# B&R Automation Studio project Sh_0218_l2
Automation Studio 4.5.2.102

## Configuration labBR

### Task classes (Cpu.sw)
```
Cyclic#4:
  DoorCtrl <- DoorCtrl.prg
  LedCtrl <- LedCtrl.prg
Binaries: TCData, udbdef, ashwd, User, asfw, arconfig, sysconf, Role, iomap, ashwac
Libraries: sys_lib, Runtime, asstring, GateCtrl, X64Lib
```

### Hardware
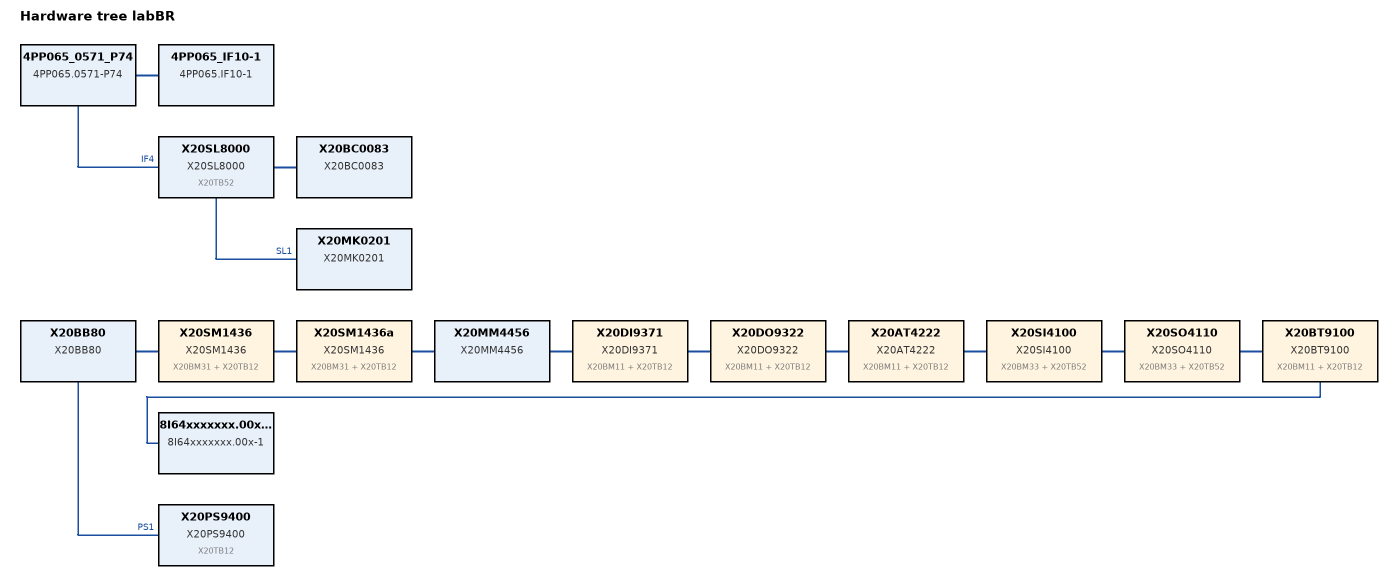
```
4PP065_0571_P74 : 4PP065.0571-P74 v1.1.2.0
  Connector IF5:
    ActivateDevice = 1
    Mode = Manual
    InternetAddress = 10.0.1.10
    SubnetMask = 255.255.255.0
  ConfigurationID = labBR
  Simulation = 1
  TimerDeviceType = EPLX2X
  TimerDevice = 4PP065_0571_P74.IF4
  TaskClassIdleTime = 2000
  Cyclic1Duration = 2000
  Cyclic1Tolerance = 0
  Cyclic1Output = 1
4PP065_IF10-1 : 4PP065.IF10-1 v1.0.3.0  [SS -> 4PP065_0571_P74.SS1]
8I64xxxxxxx.00x-1 : 8I64xxxxxxx.00x-1 v1.3.9.1  [X2X1 -> X20BT9100.X2X1 [Cable Type=X2XCable, Length=10, Version=1.0.0.2]]
  FunctionModel = Standard
  packedETAD = packed
  packedETI = packed
  packedCMDD = packed
  packedCMI = packed
  UNS = 220
  NCR = 10
  NSP = 890
  COS = 64
  RSC = 33000
X20AT4222 : X20AT4222 v1.2.3.0  [SS1 -> X20TB12e.SS; SL -> X20BM11c.SL1]
X20BB80 : X20BB80 v1.0.2.0
X20BC0083 : X20BC0083 v2.7.0.0  [PLK1 -> X20SL8000.PLK2 (NodeNumber=2) [Cable Type=PowerlinkCable, Length=10, Version=1.0.0.2]; SL -> X20BB80.SL1]
X20BM11 : X20BM11 v1.0.0.1  [X2X1 -> X20BM33a.X2X2]
X20BM11a : X20BM11 v1.0.0.1  [X2X1 -> X20MM4456.X2X2]
X20BM11b : X20BM11 v1.0.0.1  [X2X1 -> X20BM11a.X2X2]
X20BM11c : X20BM11 v1.0.0.1  [X2X1 -> X20BM11b.X2X2]
X20BM31 : X20BM31 v1.0.0.1  [X2X1 -> X20BB80.IF1]
X20BM31a : X20BM31 v1.0.0.1  [X2X1 -> X20BM31.X2X2]
X20BM33 : X20BM33 v1.0.0.4  [X2X1 -> X20BM11c.X2X2]
X20BM33a : X20BM33 v1.0.0.4  [X2X1 -> X20BM33.X2X2]
X20BT9100 : X20BT9100 v1.0.3.0  [SS1 -> X20TB12f.SS; SL -> X20BM11.SL1]
X20DI9371 : X20DI9371 v1.0.2.0  [SS1 -> X20TB12c.SS; SL -> X20BM11a.SL1]
X20DO9322 : X20DO9322 v1.0.3.0  [SS1 -> X20TB12d.SS; SL -> X20BM11b.SL1]
X20MK0201 : X20MK0201 v1.0.0.0  [SL -> X20SL8000.SL1]
X20MM4456 : X20MM4456 v1.1.5.0  [X2X1 -> X20BM31a.X2X2]
X20PS9400 : X20PS9400 v1.0.2.4  [SS1 -> X20TB12.SS; PS -> X20BB80.PS1]
X20SI4100 : X20SI4100 v1.10.1.1  [SS1 -> X20TB52.SS; SL -> X20BM33.SL1]
X20SL8000 : X20SL8000 v1.6.5.1  [PLK1 -> 4PP065_0571_P74.IF4 (NodeNumber=1) [Cable Type=PowerlinkCable, Length=10, Version=1.0.0.2]; PLK2 -> X20BC0083.PLK1 (NodeNumber=1) [Cable Type=PowerlinkCable, Length=10, Version=1.0.0.2]; SS1 -> X20TB52b.SS]
  SafeProject = SafeLOGIC-1
X20SM1436 : X20SM1436 v1.4.2.1  [SS1 -> X20TB12a.SS; SL -> X20BM31.SL1]
X20SM1436a : X20SM1436 v1.4.2.1  [SS1 -> X20TB12b.SS; SL -> X20BM31a.SL1]
X20SO4110 : X20SO4110 v1.10.1.1  [SS1 -> X20TB52a.SS; SL -> X20BM33a.SL1]
  SafeModuleID = 3
X20TB12 : X20TB12 v1.0.0.0
X20TB12a : X20TB12 v1.0.0.0
X20TB12b : X20TB12 v1.0.0.0
X20TB12c : X20TB12 v1.0.0.0
X20TB12d : X20TB12 v1.0.0.0
X20TB12e : X20TB12 v1.0.0.0
X20TB12f : X20TB12 v1.0.0.0
X20TB52 : X20TB52 v1.0.0.1
X20TB52a : X20TB52 v1.0.0.1
X20TB52b : X20TB52 v1.0.0.1
```

### IoMap.iom - 4PP065_0571_P74/IoMap.iom
```iecst
VAR_CONFIG
	::DoorCtrl:DoorBlock.sw1 AT %IX."X20DI9371".DigitalInput03;
	::DoorCtrl:DoorBlock.sw2 AT %IX."X20DI9371".DigitalInput04;
	::DoorCtrl:DoorBlock.sw3 AT %IX."X20DI9371".DigitalInput05;
	::DoorCtrl:CMD AT %QW."8I64xxxxxxx.00x-1".CMDD_Output;
	::DoorCtrl:ETAD AT %IW."8I64xxxxxxx.00x-1".ETAD_Input;
	::DoorCtrl:Speed AT %QW."8I64xxxxxxx.00x-1".LFRD_Output;
	::LedCtrl:sc0 AT %QX."X20DO9322".DigitalOutput02;
	::LedCtrl:sc1 AT %QX."X20DO9322".DigitalOutput03;
	::LedCtrl:sc2 AT %QX."X20DO9322".DigitalOutput04;
	::LedCtrl:sc3  AT %QX."X20DO9322".DigitalOutput05;
	::DoorCtrl:DoorBlock.sw0 AT %IX."X20DI9371".DigitalInput02;
	::DoorCtrl:DoorBlock.direction AT %IX."X20DI9371".DigitalInput01;
END_VAR
```

## Logical view

### Global.var
```iecst
VAR
	sw1 : BOOL := FALSE;
	sw2 : BOOL := FALSE;
	sw3 : BOOL := FALSE;
	sw0 : BOOL := FALSE;
END_VAR
```

### Program Logical/DoorCtrl

#### Variables.var
```iecst
VAR
	Close : BOOL;
	Open : BOOL;
	DoorBlock : FBGate;
	ETAD : UINT := 0;
	Speed : INT := 0;
	CMD : UINT := 0;
	LedBlock : FBLed;
END_VAR
```

#### Main.c
```c
#include <bur/plctypes.h>

#ifdef _DEFAULT_INCLUDES
	#include <AsDefault.h>
#endif

void _INIT ProgramInit(void)
{
	Open  = 0;
	Close = 0;
}

void _CYCLIC ProgramCyclic(void)
{
	Speed = DoorBlock.Speed;
	DoorBlock.DriveBlk.ETAD_Input = ETAD;
	CMD = DoorBlock.DriveBlk.CMDD_Output;
	if (Open == 1){
		DoorBlock.direction = 1;
	}
	if (Close == 1) {
		DoorBlock.direction = 0;
	}
	FBGate(&DoorBlock);
	if ((DoorBlock.State == ST_OPEN) || (DoorBlock.State == ST_CLOSE)){
		Open  = 0;
		Close = 0;
	}
	LedBlock.State = DoorBlock.State;
	FBLed(&LedBlock);
	sw0 = LedBlock.s1;
	sw1 = LedBlock.s2;
	sw2 = LedBlock.s3;
	sw3 = LedBlock.s4;

}

void _EXIT ProgramExit(void)
{

}
```

### Program Logical/LedCtrl

#### Variables.var
```iecst
VAR
	sc : FBLed := (0);
	sc0 : BOOL;
	sc1 : BOOL;
	sc2 : BOOL;
	sc3 : BOOL;
END_VAR
```

#### Main.c
```c
#include <bur/plctypes.h>

#ifdef _DEFAULT_INCLUDES
	#include <AsDefault.h>
#endif

void _INIT ProgramInit(void)
{

}

void _CYCLIC ProgramCyclic(void)
{
		sc0 = sw0;
		sc1 = sw1;
		sc2 = sw2;
		sc3 = sw3;

}

void _EXIT ProgramExit(void)
{

}
```

### Library Logical/Libraries/GateCtrl (ANSIC)
Depends on: X64Lib

#### Types.typ - Exported data types
```iecst
TYPE
	GateState :
		(
		ST_INIT := 0,
		ST_UNKNOWN := 1,
		ST_OPEN := 2,
		ST_CLOSE := 3,
		ST_ACC_POS := 4,
		ST_ACC_NEG := 5,
		ST_POS := 6,
		ST_NEG := 7,
		ST_DEC_POS := 8,
		ST_DEC_NEG := 9
		);
END_TYPE
```

#### GateCtrl.fun - Exported functions and function blocks
```iecst
FUNCTION_BLOCK FBLed
	VAR_OUTPUT
		s1 : BOOL;
		s2 : BOOL;
		s3 : BOOL;
		s4 : BOOL;
	END_VAR
	VAR_INPUT
		State : {REDUND_UNREPLICABLE} GateState;
	END_VAR
END_FUNCTION_BLOCK

{REDUND_ERROR} FUNCTION_BLOCK FBGate (* *) (*$GROUP=User,$CAT=User,$GROUPICON=User.png,$CATICON=User.png*)
	VAR_INPUT
		sw0 : BOOL; (*инпут датчиков*)
		sw1 : BOOL;
		sw2 : BOOL;
		sw3 : BOOL;
		State : {REDUND_UNREPLICABLE} GateState;
		direction : BOOL;
	END_VAR
	VAR_OUTPUT
		Speed : INT;
	END_VAR
	VAR
		DriveBlk : FBX64Inverter;
	END_VAR
END_FUNCTION_BLOCK
```

#### FBGate.c
```c
#include <bur/plctypes.h>
#ifdef __cplusplus
	extern "C"
	{
#endif
	#include "GateCtrl.h"
#ifdef __cplusplus
	};
#endif
/* TODO: Add your comment here */
void FBGate(struct FBGate* inst)
{
	switch (inst->State) {
		case ST_INIT: //
			inst->State = ST_UNKNOWN;
			break;
		case ST_UNKNOWN: //
			if ((inst->direction == 0) && (inst->sw0 == 0)){
			inst->State = ST_OPEN;
			}
			if ((inst->direction == 1) && (inst->sw0 == 1)){
				inst->State = ST_CLOSE;
			}
			break;
		case ST_OPEN: //
			inst->DriveBlk.enable = 0;
			FBX64Inverter(&inst->DriveBlk);
			inst->Speed = 0;
			FBX64Inverter(&inst->DriveBlk);
			if (inst->direction == 1){
				inst->State = ST_ACC_POS;
			}
			break;
		case ST_CLOSE:
			inst->DriveBlk.enable = 0;
			FBX64Inverter(&inst->DriveBlk);
			inst->Speed = 0;
			FBX64Inverter(&inst->DriveBlk);
			if (inst->direction == 0){
				inst->State = ST_ACC_NEG;
			}
			break;
		case ST_ACC_POS:
			inst->DriveBlk.enable = 1;
			inst->Speed = 100;
			FBX64Inverter(&inst->DriveBlk);
			if (inst->sw1){
				inst->State = ST_POS;
			}
			if (inst->direction == 0) {
				inst->State = ST_ACC_NEG;
			}
			break;
		case ST_ACC_NEG:
			inst->DriveBlk.enable = 1;
			FBX64Inverter(&inst->DriveBlk);
			inst->Speed = -100;
			if (!inst->sw2){
				inst->State = ST_NEG;
			}
			break;
		case ST_NEG:
			inst->Speed = -300;
			FBX64Inverter(&inst->DriveBlk);
			if (!inst->sw1){
				inst->State = ST_DEC_NEG;
			}
			break;
		case ST_DEC_NEG:
			inst->Speed = -100;
			FBX64Inverter(&inst->DriveBlk);
			if (!inst->sw0){
				inst->State = ST_OPEN;
			}
			break;
		case ST_DEC_POS:
			FBX64Inverter(&inst->DriveBlk);
			inst->Speed = 100;
			if (inst->sw3){
				inst->State = ST_CLOSE;
			}
			break;
		case ST_POS:
			FBX64Inverter(&inst->DriveBlk);
			inst->Speed = 300;
			if (inst->sw2){
				inst->State = ST_DEC_POS;
			}
			if (inst->direction == 0) {
				inst->State = ST_NEG;
			}
			break;
	}
}
```

#### FBLed.c
```c
#include <bur/plctypes.h>
#ifdef __cplusplus
	extern "C"
	{
#endif
	#include "GateCtrl.h"
#ifdef __cplusplus
	};
#endif
/* TODO: Add your comment here */
void FBLed(struct FBLed* inst)
{
	 BOOL timer;
	{
		/*TODO: Add your code here*/
		switch(inst->State)
		{
			case ST_INIT:
				{
					inst->s1 = 0;

					inst->s2 = 0;

					inst->s3 = 0;

					inst->s4 = 0;

					break;
				}

			case ST_UNKNOWN:
				{
					timer = !timer;
					if (timer == 1)
					{
						inst->s1 = 1;

						inst->s2 = 1;

						inst->s3 = 1;

						inst->s4 = 1;
					}
					else
					{

						inst->s1 = 0;

						inst->s2 = 0;

						inst->s3 = 0;

						inst->s4 = 0;
					}

				}

			case ST_OPEN:
				{
					inst->s1 = 0;

					inst->s2 = 0;

					inst->s3 = 0;

					inst->s4 = 0;

					break;
				}

			case ST_CLOSE:
				{

					inst->s1 = 1;

					inst->s2 = 1;

					inst->s3 = 1;

					inst->s4 = 1;

					break;
				}

			case ST_ACC_POS:
				{

					inst->s1 = 1;

					inst->s2 = 0;

					inst->s3 = 0;

					inst->s4 = 0;

					break;
				}

			case ST_ACC_NEG:
				{

					inst->s1 = 1;

					inst->s2 = 1;

					inst->s3 = 1;

					inst->s4 = 0;

					break;
				}

			case ST_NEG:
				{

					inst->s1 = 1;

					inst->s2 = 1;

					inst->s3 = 0;

					inst->s4 = 0;

					break;
				}

			case ST_DEC_NEG:
				{

					inst->s1 = 1;

					inst->s2 = 0;

					inst->s3 = 0;

					inst->s4 = 0;

					break;
				}

			case ST_DEC_POS:
				{

					inst->s1 = 1;

					inst->s2 = 1;

					inst->s3 = 1;

					inst->s4 = 0;

					break;
				}

					case ST_POS:
				{

					inst->s1 = 1;

					inst->s2 = 1;

					inst->s3 = 0;

					inst->s4 = 0;

					break;
				}
		}
	}
}
```

### Library Logical/Libraries/X64Lib

#### X64Lib.fun
```iecst
(********************************************************************
 * COPYRIGHT -- Microsoft
 ********************************************************************
 * Library: X64Lib
 * File: X64Lib.fun
 * Author: chuh
 * Created: April 02, 2015
 ********************************************************************
 * Functions and function blocks of library X64Lib
 ********************************************************************)

FUNCTION_BLOCK FBX64Inverter (*X64 Acopos Inverter Control Lib*) (*$GROUP=User*)
	VAR_INPUT
		enable : BOOL;
		ETAD_Input : UINT;
	END_VAR
	VAR_OUTPUT
		CMDD_Output : UINT;
	END_VAR
	VAR
		mask : UINT;
	END_VAR
END_FUNCTION_BLOCK
```

#### FBX64Inverter.c
```c
/********************************************************************
 * COPYRIGHT -- Microsoft
 ********************************************************************
 * Library: X64Lib
 * File: FBX64Inverter.c
 * Author: chuh
 * Created: April 02, 2015
 ********************************************************************
 * Implementation of library X64Lib
 ********************************************************************/

#include <bur/plctypes.h>
#ifdef __cplusplus
	extern "C"
	{
#endif

	#include "X64Lib.h"

#ifdef __cplusplus
	};
#endif

//***************Объявление списка состояний частотника  ********************
#define	ACPIX64_STATE_NOT_READY_TO_SWITCH_ON	0x0000 /* */
#define	ACPIX64_STATE_SWITCH_ON_DISABLED		0x0040 /* */
#define	ACPIX64_STATE_READY_TO_SWITCH_ON		0x0064 /* */
#define	ACPIX64_STATE_SWITCHED_ON				0x0021 /* */
#define	ACPIX64_STATE_OPERATION_ENABLED			0x0027 /* */
#define	ACPIX64_STATE_QUICK_STOP_ACTIVE			0x0007/* */
#define	ACPIX64_STATE_MALFUNCTION				0x0008/* */

#define	ACPIX64_CMD_DISABLE_VOLTAGE				0x0000/* */
#define	ACPIX64_CMD_SHUTDOWN					0x0006/* */
#define	ACPIX64_CMD_SWITCH_ON					0x0006/* */
#define	ACPIX64_CMD_ENABLE_OPERATION			0x000F/* */
#define ACPIX64_CMD_GO                          0x0007
#define	ACPIX64_CMD_FAULT_RESET					0x0080/* */

/* X64 Acopos Inverter Control Lib */
void FBX64Inverter(struct FBX64Inverter* inst)
{
	UINT MSK;			//Переменная для хранения входа после наложения маски
	MSK = inst->ETAD_Input & 0x006F;
	inst->mask = MSK;/* */ // маска на значащую информацию статуса частотника
	if(!inst->enable){
		inst->CMDD_Output = ACPIX64_CMD_DISABLE_VOLTAGE;		//	 Отключаем питание с двигателя насоса
	} else {
		switch(MSK)
		{
			case ACPIX64_STATE_SWITCH_ON_DISABLED:		inst->CMDD_Output = ACPIX64_CMD_SHUTDOWN;				break;
			case ACPIX64_STATE_READY_TO_SWITCH_ON:		inst->CMDD_Output = ACPIX64_CMD_SWITCH_ON;				break;
			case ACPIX64_STATE_SWITCHED_ON:				inst->CMDD_Output = ACPIX64_CMD_ENABLE_OPERATION;		break;
		}
	}
}
```

Listed in the project but not available here: Logical/Libraries/GateCtrl/Constants.var
